// LS Electric XG5000 project: 과년66_2
// 과년도(2019 하) 66회 2일차
// PLC NewPLC
// module base 0 slot 0: 입출력 모듈:XBC-DR20S (DC 24V 입력 12점, 릴레이 출력 8점)

PROGRAM NewProgram (task: 스캔 프로그램)

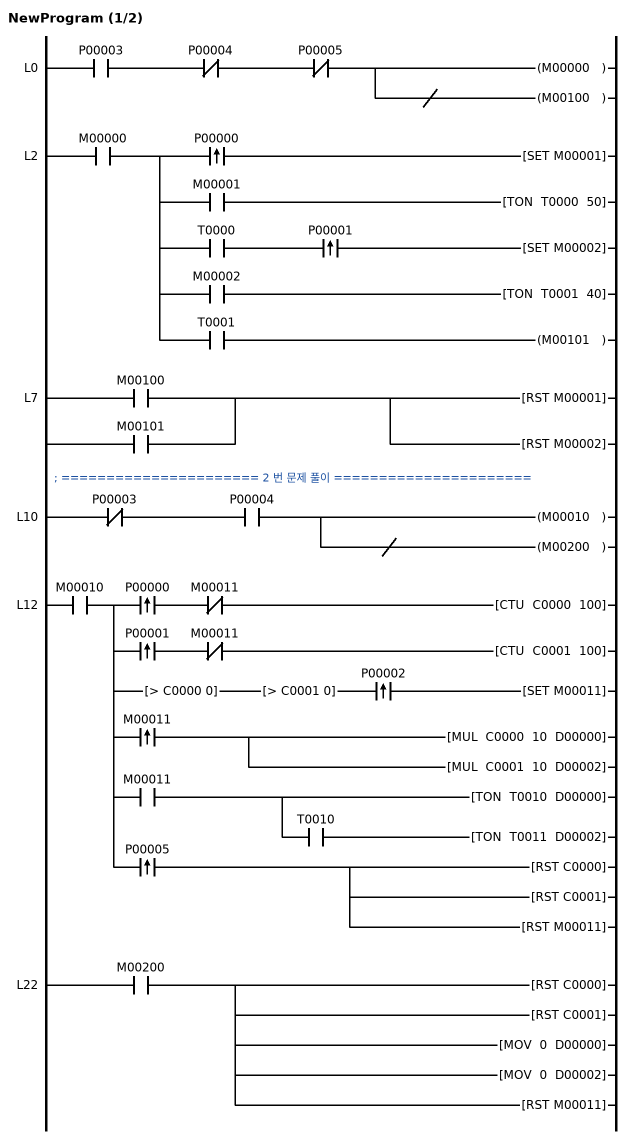
; L0
LOAD      P00003
AND NOT   P00004
AND NOT   P00005
OUT       M00000
NOT
OUT       M00100
; L2
LOAD      M00000
MPUSH
ANDP      P00000
SET       M00001
MLOAD
AND       M00001
TON       T0000 50
MLOAD
AND       T0000
ANDP      P00001
SET       M00002
MLOAD
AND       M00002
TON       T0001 40
MPOP
AND       T0001
OUT       M00101
; L7
LOAD      M00100
OR        M00101
RST       M00001
RST       M00002
// ====================== 2 번 문제 풀이 ======================
; L10
LOAD NOT  P00003
AND       P00004
OUT       M00010
NOT
OUT       M00200
; L12
LOAD      M00010
MPUSH
ANDP      P00000
AND NOT   M00011
CTU       C0000 100
MLOAD
ANDP      P00001
AND NOT   M00011
CTU       C0001 100
MLOAD
AND>      C0000 0
AND>      C0001 0
ANDP      P00002
SET       M00011
MLOAD
ANDP      M00011
MUL       C0000 10 D00000
MUL       C0001 10 D00002
MLOAD
AND       M00011
TON       T0010 D00000
AND       T0010
TON       T0011 D00002
MPOP
ANDP      P00005
RST       C0000
RST       C0001
RST       M00011
; L22
LOAD      M00200
RST       C0000
RST       C0001
MOV       0 D00000
MOV       0 D00002
RST       M00011

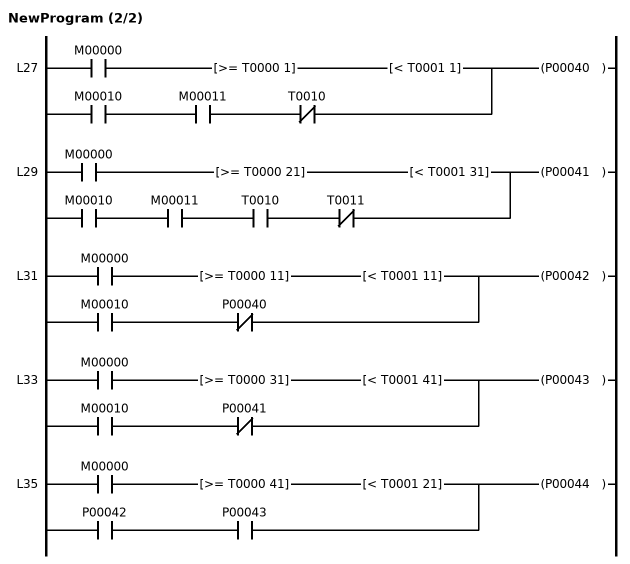
; L27
LOAD      M00000
AND>=     T0000 1
AND<      T0001 1
LOAD      M00010
AND       M00011
AND NOT   T0010
OR LOAD
OUT       P00040
; L29
LOAD      M00000
AND>=     T0000 21
AND<      T0001 31
LOAD      M00010
AND       M00011
AND       T0010
AND NOT   T0011
OR LOAD
OUT       P00041
; L31
LOAD      M00000
AND>=     T0000 11
AND<      T0001 11
LOAD      M00010
AND NOT   P00040
OR LOAD
OUT       P00042
; L33
LOAD      M00000
AND>=     T0000 31
AND<      T0001 41
LOAD      M00010
AND NOT   P00041
OR LOAD
OUT       P00043
; L35
LOAD      M00000
AND>=     T0000 41
AND<      T0001 21
LOAD      P00042
AND       P00043
OR LOAD
OUT       P00044